{attribute addProperty BoxType "EL1918-0000-0016"}
{attribute addProperty Id "FSoE_CommandUSINT811FSIN_Module_1_ErrAckBIT10.1251FSIN_Module_2_ErrAckBIT10.1251FSIN_Module_3_ErrAckBIT10.1251FSIN_Module_4_ErrAckBIT10.1251FSIN_Module_5_ErrAckBIT10.1251FSIN_Module_6_ErrAckBIT10.1251FSIN_Module_7_ErrAckBIT10.1251FSIN_Module_8_ErrAckBIT10.1251FSoE_CRC_000UINT1623FSoE_Connection_IDUINT1622"}
{attribute addProperty CRC "4068552686"}
{attribute addProperty SizeInBites "48"}
{attribute addProperty SizeInBytes "6"}
TYPE FSOE_F2812FEE :
STRUCT
	{attribute addProperty Name "FSoE_Command"}
	FSoE_Command : USINT;
	{attribute addProperty Name "FSIN_Module_1_ErrAck"}
	FSIN_Module_1_ErrAck : BIT;
	{attribute addProperty Name "FSIN_Module_2_ErrAck"}
	FSIN_Module_2_ErrAck : BIT;
	{attribute addProperty Name "FSIN_Module_3_ErrAck"}
	FSIN_Module_3_ErrAck : BIT;
	{attribute addProperty Name "FSIN_Module_4_ErrAck"}
	FSIN_Module_4_ErrAck : BIT;
	{attribute addProperty Name "FSIN_Module_5_ErrAck"}
	FSIN_Module_5_ErrAck : BIT;
	{attribute addProperty Name "FSIN_Module_6_ErrAck"}
	FSIN_Module_6_ErrAck : BIT;
	{attribute addProperty Name "FSIN_Module_7_ErrAck"}
	FSIN_Module_7_ErrAck : BIT;
	{attribute addProperty Name "FSIN_Module_8_ErrAck"}
	FSIN_Module_8_ErrAck : BIT;
	{attribute addProperty Name "FSoE_CRC_000"}
	FSoE_CRC_000 : UINT;
	{attribute addProperty Name "FSoE_Connection_ID"}
	FSoE_Connection_ID : UINT;
END_STRUCT
END_TYPE

(* stored: Version 1.2.0.0, ProductVersion 3.1.4024.9
   DUT FSOE_F2812FEE: Id {c13a28fc-ddca-4fe9-9f29-1a1d0c938bb3} *)
